FUNCTION F_Doppelmeldung : BOOL
VAR_INPUT
END_VAR
VAR
END_VAR

(* Netzwerk: 2 Doppelmeldung *)

(*
U "E1_3" E1.3 -- R Abisolierer vorn
U "E1_4" E1.4 -- R Abisolierer rück (abisoliert)
S "F45 E1.3+E1.4" M104.5 -- Doppelmeldung Abisolierer vorn+rück *)
IF GVL.insecAbisoliererIstVORN AND GVL.insecAbisoliererIstRUECK THEN
	GVL.errs.DoppelMlgAbisoVornRueck := TRUE;
END_IF


(*
U "E1_6" E1.6 -- N Crimpzange zu
U "E1_7" E1.7 -- R Crimpzange offen
S "F52 E1.6+E1.7" M105.2 -- Doppelmeldung Crimpzange zu+offen
*)
IF GVL.insecCrimpZangeIstZU AND GVL.insecCrimpZangeIstOFFEN THEN
	GVL.errs.DoppelMlgCrimpzZuOffen := TRUE;
END_IF


(*
U "E2_1" E2.1 -- R Crimpeinheit vorn
U "E2_4" E2.4 -- R Crimpeinheit rück
S "F57 E2.1+E2.4" M105.7 -- Doppelmeldung Crimpeinheit vorn+rück
*)
IF GVL.insecCrimpEinheitIstVORN AND GVL.insecCrimpEinheitIstRUECK THEN
	GVL.errs.DoppelMlgCrimpEinhVornZurueck := TRUE;
END_IF

END_FUNCTION

(* stored: Version 1.1.0.1, ProductVersion 3.1.4024.3
   POU F_Doppelmeldung: Id {c6e37c1e-2b6c-4de6-a31f-ae008768269d}, SpecialFunc None *)
